PROGRAM MAIN
VAR
END_VAR

END_PROGRAM

(* stored: Version 1.1.0.1
   POU MAIN: Id {2c2cd341-53ff-4a1d-8582-8b3c7243878f} *)
